// TIA Portal V19 export
DATA_BLOCK "ValvesScadaInfo"   // DB22
{ S7_Optimized_Access := 'TRUE' }
// stored: AutoNumber false, MemoryReserve 0
   VAR RETAIN
      V01_01 : "ValvesInfo_UDT";
      V01_03 : "ValvesInfo_UDT";
      V01_04 : "ValvesInfo_UDT";
      V01_08 : "ValvesInfo_UDT";
      V01_09 : "ValvesInfo_UDT";
      V01_11 : "ValvesInfo_UDT";
      V01_12 : "ValvesInfo_UDT";
      V01_13 : "ValvesInfo_UDT";
      V01_14 : "ValvesInfo_UDT";
      V01_15 : "ValvesInfo_UDT";
      V01_16 : "ValvesInfo_UDT";
      V01_17 : "ValvesInfo_UDT";
      V09_04 : "ValvesInfo_UDT";
      V09_05 : "ValvesInfo_UDT";
      V09_06 : "ValvesInfo_UDT";
      V09_07 : "ValvesInfo_UDT";
      V09_08 : "ValvesInfo_UDT";
      V09_09 : "ValvesInfo_UDT";
      V09_10 : "ValvesInfo_UDT";
      V09_11 : "ValvesInfo_UDT";
      V09_12 : "ValvesInfo_UDT";
   END_VAR
BEGIN
END_DATA_BLOCK
